// TIA Portal V20 export
FUNCTION "FC_ManualStopper" : Void   // FC13, LAD
// stored: Access Published, Namespace Global, SetENOAutomatically false
   VAR_INPUT
      GoUp : Bool;
      GoDown : Bool;
      positionUp : Bool;
      positionDown : Bool;
   END_VAR
   VAR_OUTPUT
      CmdUP : Bool;
      cmdDOWN : Bool;
   END_VAR
BEGIN

REGION Network 1: status manual
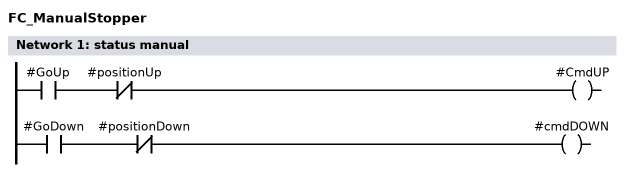
   RUNG wire#powerrail
      Contact( #GoUp )
      I_Contact( #positionUp )
      Coil( #CmdUP )
   END_RUNG
   RUNG wire#powerrail
      Contact( #GoDown )
      I_Contact( #positionDown )
      Coil( #cmdDOWN )
   END_RUNG
   // the same network as SCL:
   #CmdUP := #GoUp AND NOT #positionUp;
   #cmdDOWN := #GoDown AND NOT #positionDown;
END_REGION
END_FUNCTION
